INTERFACE PUBLIC CompletedCommands

METHOD PUBLIC Abort
END_METHOD

METHOD PUBLIC Reset
END_METHOD

METHOD PUBLIC Stop
END_METHOD

END_INTERFACE

(* stored: Version 1.1.0.1, ProductVersion 3.1.4026.12
   Itf CompletedCommands: Id {ec0323ba-8561-0e01-188f-98bb79bd5ab9}
   Method Abort: Id {8c73f3a8-9652-4614-8fca-234b6c8262dd}
   Method Reset: Id {0a3bd21e-210b-0b21-2287-f384442eb68d}
   Method Stop: Id {0c556ba7-3b95-4c19-9c7d-95c4dc8626b1} *)
